// TwinCAT 3 PLC project PlcTurntable
// ProgramVersion: 3.1.4024.0
// libraries:
//   Tc2_System, * (Beckhoff Automation GmbH)
// project tree:
//   POUs/ F_DegreesToRadians.TcPOU, MAIN.TcPOU
// real-time tasks:
//   TASK PlcTask: cycle T#10ms, priority 20, ADS port 350

// ---- POUs/F_DegreesToRadians.TcPOU
FUNCTION F_DegreesToRadians : LREAL
VAR_INPUT
    degrees : LREAL;
END_VAR
VAR CONSTANT
    d2r : LREAL := PI/180.0;
END_VAR

F_DegreesToRadians := degrees * d2r;

END_FUNCTION

// ---- POUs/MAIN.TcPOU
PROGRAM MAIN
VAR
    commandedDegPerSec : LREAL;
    commandedRadPerSec : LREAL;
END_VAR

commandedDegPerSec := 15.0;
commandedRadPerSec := F_DegreesToRadians(degrees := commandedDegPerSec);

END_PROGRAM
